// TwinCAT 3 PLC project L2SIVacuum
// Title: LCLS Vacuum
// Company: SLAC - LCLS
// Author: LCLS ECS-Platforms
// ProjectVersion: 0.0.0
// ProgramVersion: 3.1.4020.5
// libraries:
//   LCLS General, * (SLAC)
//   LCLSVacuumSerialDriverLib, * (SLAC - LCLS)
//   PMPS, * (SLAC - LCLS)
//   Tc2_DataExchange, * (Beckhoff Automation GmbH)
//   Tc2_EtherCAT, * (Beckhoff Automation GmbH)
//   Tc2_ModbusSrv, * (Beckhoff Automation GmbH)
//   Tc2_Standard, * (Beckhoff Automation GmbH)
//   Tc2_System, * (Beckhoff Automation GmbH)
//   Tc2_TcpIp, * (Beckhoff Automation GmbH)
//   Tc2_Utilities, * (Beckhoff Automation GmbH)
//   Tc3_EventLogger, * (Beckhoff Automation GmbH)
//   Tc3_JsonXml, * (Beckhoff Automation GmbH)
//   Tc3_Module, * (Beckhoff Automation GmbH)
//   TcUnit, * (www.tcunit.org)
// project tree:
//   DUTs/Gauges/ E_PressureState.TcDUT (not stored), Gauge_Type.TcDUT (not stored), ST_VG.TcDUT (not stored)
//   DUTs/Pumps/ E_PumpState.TcDUT (not stored), ST_AgilentPTM.TcDUT (not stored), ST_EbaraDryPump.TcDUT (not stored), ST_EbaraEVA.TcDUT (not stored), ST_EbaraPTM.TcDUT (not stored), ST_KashiyamaDryPump.TcDUT (not stored), ST_LeyboldPTM.TcDUT (not stored), ST_PfeifferPTM.TcDUT (not stored), ST_PIP.TcDUT (not stored), ST_PTM.TcDUT (not stored), ST_RoughPump.TcDUT (not stored)
//   DUTs/Valves/ E_ValvePositionState.TcDUT (not stored), E_VCN.TcDUT (not stored), E_VGC.TcDUT (not stored), ST_ValveBase.TcDUT (not stored), ST_VFS.TcDUT (not stored), ST_VGC_2S.TcDUT (not stored), ST_VRC_NO.TcDUT (not stored), ST_VWC_NO.TcDUT (not stored), ST_VVC.TcDUT (not stored), ST_VCC_NO.TcDUT (not stored), ST_VCN.TcDUT (not stored), ST_VGC.TcDUT (not stored), ST_VRC.TcDUT (not stored)
//   GVLs/ Constants.TcGVL (not stored), Global_Variables.TcGVL (not stored)
//   / PlcTask.TcTTO (not stored)
//   POUs/ADS/ FB_ADS.TcPOU (not stored), FB_ADS_WATCHDOG.TcPOU (not stored), FB_TBOOL_ADS.TcPOU (not stored)
//   POUs/Functions/Deprecated/Gauges/ FB_MKS317A.TcPOU (not stored), FB_MKS500_EP.TcPOU (not stored), FB_PressureState.TcPOU (not stored)
//   POUs/Functions/Deprecated/Valves/ FB_VCC.TcPOU (not stored), FB_VCC_NO.TcPOU (not stored), FB_VGC_AP.TcPOU (not stored), FB_VGC_EBD.TcPOU (not stored)
//   POUs/Functions/Gauges/ FB_901_ECAT.TcPOU (not stored), FB_9XX.TcPOU (not stored), FB_972.TcPOU (not stored), FB_GaugeBase.TcPOU (not stored), FB_CVM201.TcPOU (not stored), FB_CCM501.TcPOU (not stored), FB_IE514.TcPOU, FB_MKS909.TcPOU (not stored), FB_CMR362.TcPOU (not stored), FB_GCM.TcPOU (not stored), FB_ITR90.TcPOU (not stored), FB_MKS392.TcPOU (not stored), FB_MKS500.TcPOU (not stored), FB_MKS722.TcPOU (not stored), FB_MKS_937A.TcPOU (not stored), FB_MKS317.TcPOU (not stored), FB_MKS275.TcPOU (not stored), FB_MKS_937B.TcPOU (not stored), FB_MKS422.TcPOU (not stored)
//   POUs/Functions/Gauges/Interfaces/ FB_GaugeModbus.TcPOU (not stored), FB_Gauge_Interface.TcPOU (not stored), FB_TGCC_ADS.TcPOU (not stored), FB_TGPI_ADS.TcPOU (not stored)
//   POUs/Functions/Pumps/ FB_EbaraDryPump.TcPOU (not stored), FB_EbaraEVA.TcPOU (not stored), FB_KashiyamaPump.TcPOU (not stored), FB_PIP_Gamma.TcPOU (not stored), FB_PIP_SIP.TcPOU (not stored), FB_PTM_Agilent.TcPOU (not stored), FB_PTM_Ebara_011M.TcPOU (not stored), FB_PTM_Ebara_010M.TcPOU (not stored), FB_PTM_MagDriveDigital.TcPOU (not stored), FB_PTM_Pfeiffer.TcPOU (not stored), FB_PTM_TurboDrive.TcPOU (not stored), FB_PTM_TwisTorr.TcPOU (not stored), FB_Pump.TcPOU (not stored), FB_ScrollPump.TcPOU (not stored)
//   POUs/Functions/Pumps/functions/ FB_TurboExtLogic.TcPOU (not stored), F_TurboExtILK_NO.TcPOU (not stored), F_TurboExtILKLogic.TcPOU (not stored), F_TurboExtILKLogic_2.TcPOU (not stored), F_TurboExtILK_NO_1.TcPOU (not stored)
//   POUs/Functions/Pumps/Interfaces/ FB_PIP_Interface_In.TcPOU (not stored), FB_PIP_Interface_Out.TcPOU (not stored), FB_TPIP_ADS.TcPOU (not stored)
//   POUs/Functions/Valves/ FB_Kashiyama_VRC.TcPOU (not stored), FB_MKS248.TcPOU (not stored), FB_TurbVentvalve_NO.TcPOU (not stored), FB_Valve.TcPOU (not stored), FB_VFS.TcPOU (not stored), FB_VGC_2S.TcPOU (not stored), FB_VRC_DA.TcPOU (not stored), FB_VRC_EBD.TcPOU (not stored), FB_VRC_NO.TcPOU (not stored), FB_VRC_NO_FFO.TcPOU (not stored), FB_VVC.TcPOU (not stored), FB_VCN.TcPOU (not stored), FB_VGC.TcPOU (not stored), FB_VRC.TcPOU (not stored), FB_VRC_OK_CLS.TcPOU (not stored)
//   POUs/Functions/Valves/functions/ F_RoughPumpInlet_ILK.TcPOU (not stored), F_TurboGateValve_ILK.TcPOU (not stored), F_TurboGateValve_ILK_1.TcPOU (not stored), F_TurboGateValve_Protection_ILK.TcPOU (not stored), F_TURBO_VRC_ILK.TcPOU (not stored), F_VALVE_REL_ILK.TcPOU (not stored), F_VRC_DIODE_ILK_OK.TcPOU (not stored), F_VRC_DIODE_ILK.TcPOU (not stored)
//   POUs/Functions/Valves/Interfaces/ FB_TVGC_2S_ADS.TcPOU (not stored), FB_VFS_Interface.TcPOU (not stored), FB_TVGC_ADS.TcPOU (not stored), FB_Valve_Interface.TcPOU (not stored), ITF_Valve.TcIO (not stored)
//   UnitTests/Functions/ V_TO_INT.TcPOU (not stored)
//   UnitTests/Gauges/ FB_GCC_Test.TcPOU (not stored), FB_GPI_Test.TcPOU (not stored)
//   UnitTests/ PRG_Test.TcPOU (not stored)
//   UnitTests/Pumps/ FB_PIP_Test.TcPOU (not stored), FB_PTM_Test.TcPOU (not stored)
//   UnitTests/Valves/ FB_VGC_Test.TcPOU (not stored), FB_VRC_Test.TcPOU (not stored)
//   Version/ Global_Version.TcGVL (not stored)

// ---- POUs/Functions/Gauges/FB_IE514.TcPOU
(* This function is for the Hot Cathode IE514 connected to n IM540 *)
(*This function provides ILK and Set Point Protection for the Hot Cathode*)
FUNCTION_BLOCK FB_IE514 EXTENDS FB_GaugeBase
VAR_IN_OUT
		
END_VAR
VAR_INPUT
		PG	:	ST_VG; 
END_VAR
VAR_OUTPUT
	{attribute 'pytmc' := '
    pv: 
	'}
	IG : ST_VG; 
END_VAR
VAR
	rV	:	REAL;
	timer:TON;
	rMaxPressure	:	REAL := 7.5E-5; //Torr
	rMinPressure	:	REAL := 7.5E-14; //Torr
	
	//rDefaultVAC_SP: REAL := 9E-3; // as per manual
	
	iTermBits: UINT := 30518 ; // The terminal's maximum value in bits default el3174 as per vacuum architecture
	(*IOs to be linked*)
	/// Controls and I/Os
	i_iPRESS_R AT %I* :INT; // input Pressure // Link to analog Input
	q_xHV_DIS AT %Q* : BOOL := True; // Disable Gauge High Voltage when True // 'TcLinkTo' (EL2794) ^Output
	i_xHV_ON AT %I*	: BOOL; //  True when High Voltage is on  // 'TcLinkTo' (EL1124) ^Input
END_VAR

(* 6-xx-2021, Patrick Ayers *)
(* This function will read the pressure from an IE514 gauge on an IM540. *)

(*Soft IO Linking*)
IO();

(*Pressure readbacks*)
// check no div by zero
If (iTermBits=0) THEN iTermBits := 30518;END_IF
rV := 10*INT_TO_REAL(IG.i_iPRESS_R)/iTermBits;

//conversion
IG.rPRESS := LREAL_TO_REAL(EXPT(10, rV));	//manual page 70 IM540 (Mode Full)

(* Pressure gauge State checks *)
IF (rV <=10) AND (rV>0) THEN
	IG.eState := Valid; // normal
ELSIF rV >= 0.18 AND rV <= 0.22 THEN 
	IG.eState := ValidLo; //LO
ELSIF rV > 9.6 AND rV<= 9.9 THEN
	IG.eState := ValidHi; //HIGH
ELSIF rV <= 0 THEN // 
	IG.eState := GaugeDisconnected; //not on
	IG.rPRESS :=rMinPressure;
ELSE
	IG.eState := PressInvalid; //other fault - could be no gauge, controller powering up etc
	IG.rPRESS := 0;
END_IF


(* Ion Gauge Protection Functions *)
(* If the PG pressure is greater than the VG.PRO_SP then the gauge is disabled *)
(* If the PG pressure is less than the VG.PRO_SP then the gauge is enabled *)
(* This FB also implements some hysteresis so the gauge doesn't have rapid power cycling while near the turn on boundary *)

	IF (PG.rPRESS <= IG.rPRO_SP) THEN
		 IG.q_xHV_DIS := NOT IG.xHV_SW;
		 IG.xILKOk := TRUE;
	ELSIF NOT IG.q_xHV_DIS AND timer.Q THEN
		IF IG.rPRESS > (IG.rPRO_SP + IG.rHYS_PR) OR PG.rPRESS > (IG.rPRO_SP + IG.rHYS_PR) THEN
		IG.q_xHV_DIS := TRUE;
		IG.xHV_SW := FALSE;
		END_IF
	ELSE 
		IG.q_xHV_DIS := TRUE;
		IG.xHV_SW := FALSE;
		IG.xILKOk := FALSE;
 	END_IF
 


 
(* Pressure gauge OK checks *)
IG.xPRESS_OK := (rV <=10) AND (rV>0);


(* Setpoint evaluation *)
IG.xAT_VAC := IG.xPRESS_OK AND IG.rPRESS < IG.rVAC_SP;


(*Logger*)
ACT_Logger();
(*Soft IO Linking*)
// check ethercat Diagnostics
IO();
(*Load or save the persistent variables*)
ACT_Persistent();
timer(IN:= NOT IG.q_xHV_DIS, PT:= T#2s);

ACTION ACT_Logger:
// ILK logger
IF (IG.xLog) THEN
	IF NOT IG.xILKOk AND NOT IG.q_xHV_DIS THEN
			fbLogger(sMsg:='Lost external interlock while gauge was on.', eSevr:=TcEventSeverity.Critical);  	
	END_IF
	
	
	// Log Action
	tAction(CLK:=  IG.xHV_SW);
	IF tAction.Q THEN fbLogger(sMsg:='Ion gauge commanded to switch on', eSevr:=TcEventSeverity.Info); END_IF
	
	
	
	//STATE Logger  
	IF ePrevState <> IG.eState THEN
		  CASE IG.eState OF
			ValidHi:
				fbLogger(sMsg:='Gauge pressure valid high.', eSevr:=TcEventSeverity.Info);
			ValidLo:
				fbLogger(sMsg:='Gauge pressure valid low.', eSevr:=TcEventSeverity.Info);
			Valid:
				fbLogger(sMsg:='Gauge pressure valid.', eSevr:=TcEventSeverity.Info);
			GaugeDisconnected:
				fbLogger(sMsg:='Gauge Disconnected.', eSevr:=TcEventSeverity.Critical);
			PressInvalid:
				fbLogger(sMsg:='Gauge pressure invalid.', eSevr:=TcEventSeverity.Warning);
			OoR:
				fbLogger(sMsg:='Gauge pressure out of range.', eSevr:=TcEventSeverity.Warning);
			Starting:
				fbLogger(sMsg:='Gauge starting.', eSevr:=TcEventSeverity.Info);
		  END_CASE
		  ePrevState := IG.eState;  
	  END_IF
END_IF
END_ACTION

ACTION ACT_Persistent:
(*On first PLC pass, load the persistent value into the structrue variable*)
IF (SUPER^.bRestorePersistentData) THEN
	SUPER^.bRestorePersistentData	:= FALSE;
	IF ( rVAC_SP <> 0) THEN
		IG.rVAC_SP := rVAC_SP;
	END_IF;
	IF ( rPRO_SP <> 0) THEN
		IG.rPRO_SP := rPRO_SP;
	END_IF;
	IF ( rHYS_PR <> 0) THEN
		IG.rHYS_PR := rHYS_PR;
	END_IF;
END_IF
(*Check if a new value has been written in the structure variable copy it to the persistent variable*)
IF NOT (IG.rVAC_SP = rVAC_SP)  THEN
	rVAC_SP := IG.rVAC_SP;
END_IF;

IF NOT (IG.rPRO_SP = rPRO_SP) THEN
	rPRO_SP:= IG.rPRO_SP;
END_IF;

IF NOT (IG.rHYS_PR = rHYS_PR) THEN
	rHYS_PR:= IG.rHYS_PR;
END_IF;
END_ACTION

ACTION IO:
(*soft link inputs*)
IG.i_iPRESS_R:=	i_iPRESS_R; 

(*soft link outputs*)
q_xHV_DIS := IG.q_xHV_DIS;

IG.i_xHV_ON:= i_xHV_ON;

IG.sPath := sPath;
END_ACTION

METHOD M_AutoOn : BOOL
VAR_INPUT
END_VAR
this^.IG.q_xHV_DIS:= FALSE;
END_METHOD

METHOD M_HVE : BOOL
VAR_INPUT
		enable:bool; // set to true to enable, false to disable;
END_VAR

this^.IG.xHV_SW:= (enable);
END_METHOD

END_FUNCTION_BLOCK
